
FUNCTION CB_sint_to_word : WORD

TITLE = ' Convert an integer into a word '
VERSION : '1.0'
AUTHOR  : CB
NAME    : sinToWor
FAMILY  : TNI

VAR_INPUT
    IN : INT;
END_VAR

BEGIN

CB_sint_to_word := BYTE_TO_WORD(INT_TO_BYTE(IN));

END_FUNCTION
